{attribute addProperty BoxType "EK1100-0000-0018"}
{attribute addProperty Id "Beckhoff_EL72xxEK1122Beckhoff_EL72xxEK1122_DA7F4B70162A_0001_EL7201_0000_0017EL7201_83D4128E25031.25A_0002_EL7201_0000_0018EL7201_83D4128E25031.25A_0003_EL7201_0000_0019EL7201_83D4128E25031.25A_0004_EL7201_0000_0020EL7201_83D4128E25031.25A_0005_EL7201_0000_0021EL7201_83D4128E25031.25A_0006_EL7201_0001_0017EL7201_789C0F5925031.25A_0007_EL7201_0001_0018EL7201_789C0F5925031.25A_0008_EL7201_0001_0019EL7201_789C0F5925031.25A_0009_EL7201_0001_0020EL7201_789C0F5925031.25A_0010_EL7201_0001_0021EL7201_789C0F5925031.25A_0011_EL7201_0010_0019EL7201_83D4128E25031.25A_0012_EL7201_0010_0020EL7201_83D4128E25031.25A_0013_EL7201_0010_0021EL7201_83D4128E25031.25A_0014_EL7201_0010_0022EL7201_83D4128E25031.25A_0015_EL7201_0010_0023EL7201_83D4128E25031.25A_0016_EL7201_0010_0024EL7201_83D4128E25031.25A_0017_EL7201_0010_0025EL7201_83D4128E25031.25A_0018_EL7201_0010_0026EL7201_83D4128E25031.25A_0019_EL7201_0010_0027EL7201_83D4128E25031.25A_0020_EL7201_0010_0028EL7201_83D4128E25031.25A_0021_EL7201_0010_0029EL7201_83D4128E25031.25A_0022_EL7201_0010_0030EL7201_2D7B43DC25832.25A_0023_EL7201_0010_0031EL7201_2D7B43DC25832.25A_0024_EL7201_0010_0032EL7201_2D7B43DC25832.25A_0025_EL7201_0011_0019EL7201_789C0F5925031.25A_0026_EL7201_0011_0020EL7201_789C0F5925031.25A_0027_EL7201_0011_0021EL7201_789C0F5925031.25A_0028_EL7201_0011_0022EL7201_789C0F5925031.25A_0029_EL7201_0011_0023EL7201_789C0F5925031.25A_0030_EL7201_0011_0024EL7201_789C0F5925031.25A_0031_EL7201_0011_0025EL7201_789C0F5925031.25A_0032_EL7201_0011_0026EL7201_789C0F5925031.25A_0033_EL7201_0011_0027EL7201_789C0F5925031.25A_0034_EL7201_0011_0028EL7201_789C0F5925031.25A_0035_EL7201_0011_0029EL7201_789C0F5925031.25A_0036_EL7201_0011_0030EL7201_789C0F5925031.25A_0037_EL7201_0011_0031EL7201_789C0F5925031.25A_0038_EL7201_0011_0032EL7201_789C0F5925031.25A_0039_EL7211_0000_0020EL7211_83D4128E25031.25A_0040_EL7211_0000_0021EL7211_83D4128E25031.25A_0041_EL7211_0001_0020EL7211_789C0F5925031.25A_0042_EL7211_0001_0021EL7211_789C0F5925031.25A_0043_EL7211_0010_0023EL7211_83D4128E25031.25A_0044_EL7211_0010_0024EL7211_83D4128E25031.25A_0045_EL7211_0010_0025EL7211_83D4128E25031.25A_0046_EL7211_0010_0026EL7211_83D4128E25031.25A_0047_EL7211_0010_0027EL7211_83D4128E25031.25A_0048_EL7211_0010_0028EL7211_83D4128E25031.25A_0049_EL7211_0010_0029EL7211_83D4128E25031.25A_0050_EL7211_0010_0030EL7211_2D7B43DC25832.25A_0051_EL7211_0010_0031EL7211_2D7B43DC25832.25A_0052_EL7211_0010_0032EL7211_2D7B43DC25832.25A_0053_EL7211_0011_0023EL7211_789C0F5925031.25A_0054_EL7211_0011_0024EL7211_789C0F5925031.25A_0055_EL7211_0011_0025EL7211_789C0F5925031.25A_0056_EL7211_0011_0026EL7211_789C0F5925031.25A_0057_EL7211_0011_0027EL7211_789C0F5925031.25A_0058_EL7211_0011_0028EL7211_789C0F5925031.25A_0059_EL7211_0011_0029EL7211_789C0F5925031.25A_0060_EL7211_0011_0030EL7211_789C0F5925031.25A_0061_EL7211_0011_0031EL7211_789C0F5925031.25A_0062_EL7211_0011_0032EL7211_789C0F5925031.25A_0063_EL7201_9014_0026EL7201_83D4128E25031.25A_0064_EL7201_9014_0027EL7201_83D4128E25031.25A_0065_EL7201_9014_0028EL7201_83D4128E25031.25A_0066_EL7201_9014_0029EL7201_83D4128E25031.25A_0067_EL7201_9014_0030EL7201_2D7B43DC25832.25A_0068_EL7201_9014_0031EL7201_2D7B43DC25832.25A_0069_EL7201_9014_0032EL7201_2D7B43DC25832.25A_0070_EL7201_9015_0026EL7201_789C0F5925031.25A_0071_EL7201_9015_0027EL7201_789C0F5925031.25A_0072_EL7201_9015_0028EL7201_789C0F5925031.25A_0073_EL7201_9015_0029EL7201_789C0F5925031.25A_0074_EL7201_9015_0030EL7201_789C0F5925031.25A_0075_EL7201_9015_0031EL7201_789C0F5925031.25A_0076_EL7201_9015_0032EL7201_789C0F5925031.25A_0077_EL7211_9014_0026EL7211_83D4128E25031.25A_0078_EL7211_9014_0027EL7211_83D4128E25031.25A_0079_EL7211_9014_0028EL7211_83D4128E25031.25A_0080_EL7211_9014_0029EL7211_83D4128E25031.25A_0081_EL7211_9014_0030EL7211_2D7B43DC25832.25A_0082_EL7211_9014_0031EL7211_2D7B43DC25832.25A_0083_EL7211_9014_0032EL7211_2D7B43DC25832.25A_0084_EL7211_9015_0026EL7211_789C0F5925031.25A_0085_EL7211_9015_0027EL7211_789C0F5925031.25A_0086_EL7211_9015_0028EL7211_789C0F5925031.25A_0087_EL7211_9015_0029EL7211_789C0F5925031.25A_0088_EL7211_9015_0030EL7211_789C0F5925031.25A_0089_EL7211_9015_0031EL7211_789C0F5925031.25A_0090_EL7211_9015_0032EL7211_789C0F5925031.25A_0091_EL7221_0000_0021EL7221_83D4128E25031.25A_0092_EL7221_0001_0021EL7221_789C0F5925031.25A_0093_EL7221_9014_0028EL7221_83D4128E25031.25A_0094_EL7221_9014_0029EL7221_83D4128E25031.25A_0095_EL7221_9014_0030EL7221_2D7B43DC25832.25A_0096_EL7221_9014_0031EL7221_2D7B43DC25832.25A_0097_EL7221_9014_0032EL7221_2D7B43DC25832.25A_0098_EL7221_9015_0028EL7221_789C0F5925031.25A_0099_EL7221_9015_0029EL7221_789C0F5925031.25A_0100_EL7221_9015_0030EL7221_789C0F5925031.25A_0101_EL7221_9015_0031EL7221_789C0F5925031.25A_0102_EL7221_9015_0032EL7221_789C0F5925031.25"}
{attribute addProperty CRC "2978563334"}
{attribute addProperty SizeInBites "25636"}
{attribute addProperty SizeInBytes "3204.5"}
TYPE Beckhoff_EL72xx_B1894506 EXTENDS EK1100_179A0949 :
STRUCT
	{attribute addProperty Name "Beckhoff_EL72xxEK1122"}
	Beckhoff_EL72xxEK1122 : Beckhoff_EL72xxEK1122_DA7F4B70;
	{attribute addProperty Name "A_0001_EL7201_0000_0017"}
	A_0001_EL7201_0000_0017 : EL7201_83D4128E;
	{attribute addProperty Name "A_0002_EL7201_0000_0018"}
	A_0002_EL7201_0000_0018 : EL7201_83D4128E;
	{attribute addProperty Name "A_0003_EL7201_0000_0019"}
	A_0003_EL7201_0000_0019 : EL7201_83D4128E;
	{attribute addProperty Name "A_0004_EL7201_0000_0020"}
	A_0004_EL7201_0000_0020 : EL7201_83D4128E;
	{attribute addProperty Name "A_0005_EL7201_0000_0021"}
	A_0005_EL7201_0000_0021 : EL7201_83D4128E;
	{attribute addProperty Name "A_0006_EL7201_0001_0017"}
	A_0006_EL7201_0001_0017 : EL7201_789C0F59;
	{attribute addProperty Name "A_0007_EL7201_0001_0018"}
	A_0007_EL7201_0001_0018 : EL7201_789C0F59;
	{attribute addProperty Name "A_0008_EL7201_0001_0019"}
	A_0008_EL7201_0001_0019 : EL7201_789C0F59;
	{attribute addProperty Name "A_0009_EL7201_0001_0020"}
	A_0009_EL7201_0001_0020 : EL7201_789C0F59;
	{attribute addProperty Name "A_0010_EL7201_0001_0021"}
	A_0010_EL7201_0001_0021 : EL7201_789C0F59;
	{attribute addProperty Name "A_0011_EL7201_0010_0019"}
	A_0011_EL7201_0010_0019 : EL7201_83D4128E;
	{attribute addProperty Name "A_0012_EL7201_0010_0020"}
	A_0012_EL7201_0010_0020 : EL7201_83D4128E;
	{attribute addProperty Name "A_0013_EL7201_0010_0021"}
	A_0013_EL7201_0010_0021 : EL7201_83D4128E;
	{attribute addProperty Name "A_0014_EL7201_0010_0022"}
	A_0014_EL7201_0010_0022 : EL7201_83D4128E;
	{attribute addProperty Name "A_0015_EL7201_0010_0023"}
	A_0015_EL7201_0010_0023 : EL7201_83D4128E;
	{attribute addProperty Name "A_0016_EL7201_0010_0024"}
	A_0016_EL7201_0010_0024 : EL7201_83D4128E;
	{attribute addProperty Name "A_0017_EL7201_0010_0025"}
	A_0017_EL7201_0010_0025 : EL7201_83D4128E;
	{attribute addProperty Name "A_0018_EL7201_0010_0026"}
	A_0018_EL7201_0010_0026 : EL7201_83D4128E;
	{attribute addProperty Name "A_0019_EL7201_0010_0027"}
	A_0019_EL7201_0010_0027 : EL7201_83D4128E;
	{attribute addProperty Name "A_0020_EL7201_0010_0028"}
	A_0020_EL7201_0010_0028 : EL7201_83D4128E;
	{attribute addProperty Name "A_0021_EL7201_0010_0029"}
	A_0021_EL7201_0010_0029 : EL7201_83D4128E;
	{attribute addProperty Name "A_0022_EL7201_0010_0030"}
	A_0022_EL7201_0010_0030 : EL7201_2D7B43DC;
	{attribute addProperty Name "A_0023_EL7201_0010_0031"}
	A_0023_EL7201_0010_0031 : EL7201_2D7B43DC;
	{attribute addProperty Name "A_0024_EL7201_0010_0032"}
	A_0024_EL7201_0010_0032 : EL7201_2D7B43DC;
	{attribute addProperty Name "A_0025_EL7201_0011_0019"}
	A_0025_EL7201_0011_0019 : EL7201_789C0F59;
	{attribute addProperty Name "A_0026_EL7201_0011_0020"}
	A_0026_EL7201_0011_0020 : EL7201_789C0F59;
	{attribute addProperty Name "A_0027_EL7201_0011_0021"}
	A_0027_EL7201_0011_0021 : EL7201_789C0F59;
	{attribute addProperty Name "A_0028_EL7201_0011_0022"}
	A_0028_EL7201_0011_0022 : EL7201_789C0F59;
	{attribute addProperty Name "A_0029_EL7201_0011_0023"}
	A_0029_EL7201_0011_0023 : EL7201_789C0F59;
	{attribute addProperty Name "A_0030_EL7201_0011_0024"}
	A_0030_EL7201_0011_0024 : EL7201_789C0F59;
	{attribute addProperty Name "A_0031_EL7201_0011_0025"}
	A_0031_EL7201_0011_0025 : EL7201_789C0F59;
	{attribute addProperty Name "A_0032_EL7201_0011_0026"}
	A_0032_EL7201_0011_0026 : EL7201_789C0F59;
	{attribute addProperty Name "A_0033_EL7201_0011_0027"}
	A_0033_EL7201_0011_0027 : EL7201_789C0F59;
	{attribute addProperty Name "A_0034_EL7201_0011_0028"}
	A_0034_EL7201_0011_0028 : EL7201_789C0F59;
	{attribute addProperty Name "A_0035_EL7201_0011_0029"}
	A_0035_EL7201_0011_0029 : EL7201_789C0F59;
	{attribute addProperty Name "A_0036_EL7201_0011_0030"}
	A_0036_EL7201_0011_0030 : EL7201_789C0F59;
	{attribute addProperty Name "A_0037_EL7201_0011_0031"}
	A_0037_EL7201_0011_0031 : EL7201_789C0F59;
	{attribute addProperty Name "A_0038_EL7201_0011_0032"}
	A_0038_EL7201_0011_0032 : EL7201_789C0F59;
	{attribute addProperty Name "A_0039_EL7211_0000_0020"}
	A_0039_EL7211_0000_0020 : EL7211_83D4128E;
	{attribute addProperty Name "A_0040_EL7211_0000_0021"}
	A_0040_EL7211_0000_0021 : EL7211_83D4128E;
	{attribute addProperty Name "A_0041_EL7211_0001_0020"}
	A_0041_EL7211_0001_0020 : EL7211_789C0F59;
	{attribute addProperty Name "A_0042_EL7211_0001_0021"}
	A_0042_EL7211_0001_0021 : EL7211_789C0F59;
	{attribute addProperty Name "A_0043_EL7211_0010_0023"}
	A_0043_EL7211_0010_0023 : EL7211_83D4128E;
	{attribute addProperty Name "A_0044_EL7211_0010_0024"}
	A_0044_EL7211_0010_0024 : EL7211_83D4128E;
	{attribute addProperty Name "A_0045_EL7211_0010_0025"}
	A_0045_EL7211_0010_0025 : EL7211_83D4128E;
	{attribute addProperty Name "A_0046_EL7211_0010_0026"}
	A_0046_EL7211_0010_0026 : EL7211_83D4128E;
	{attribute addProperty Name "A_0047_EL7211_0010_0027"}
	A_0047_EL7211_0010_0027 : EL7211_83D4128E;
	{attribute addProperty Name "A_0048_EL7211_0010_0028"}
	A_0048_EL7211_0010_0028 : EL7211_83D4128E;
	{attribute addProperty Name "A_0049_EL7211_0010_0029"}
	A_0049_EL7211_0010_0029 : EL7211_83D4128E;
	{attribute addProperty Name "A_0050_EL7211_0010_0030"}
	A_0050_EL7211_0010_0030 : EL7211_2D7B43DC;
	{attribute addProperty Name "A_0051_EL7211_0010_0031"}
	A_0051_EL7211_0010_0031 : EL7211_2D7B43DC;
	{attribute addProperty Name "A_0052_EL7211_0010_0032"}
	A_0052_EL7211_0010_0032 : EL7211_2D7B43DC;
	{attribute addProperty Name "A_0053_EL7211_0011_0023"}
	A_0053_EL7211_0011_0023 : EL7211_789C0F59;
	{attribute addProperty Name "A_0054_EL7211_0011_0024"}
	A_0054_EL7211_0011_0024 : EL7211_789C0F59;
	{attribute addProperty Name "A_0055_EL7211_0011_0025"}
	A_0055_EL7211_0011_0025 : EL7211_789C0F59;
	{attribute addProperty Name "A_0056_EL7211_0011_0026"}
	A_0056_EL7211_0011_0026 : EL7211_789C0F59;
	{attribute addProperty Name "A_0057_EL7211_0011_0027"}
	A_0057_EL7211_0011_0027 : EL7211_789C0F59;
	{attribute addProperty Name "A_0058_EL7211_0011_0028"}
	A_0058_EL7211_0011_0028 : EL7211_789C0F59;
	{attribute addProperty Name "A_0059_EL7211_0011_0029"}
	A_0059_EL7211_0011_0029 : EL7211_789C0F59;
	{attribute addProperty Name "A_0060_EL7211_0011_0030"}
	A_0060_EL7211_0011_0030 : EL7211_789C0F59;
	{attribute addProperty Name "A_0061_EL7211_0011_0031"}
	A_0061_EL7211_0011_0031 : EL7211_789C0F59;
	{attribute addProperty Name "A_0062_EL7211_0011_0032"}
	A_0062_EL7211_0011_0032 : EL7211_789C0F59;
	{attribute addProperty Name "A_0063_EL7201_9014_0026"}
	A_0063_EL7201_9014_0026 : EL7201_83D4128E;
	{attribute addProperty Name "A_0064_EL7201_9014_0027"}
	A_0064_EL7201_9014_0027 : EL7201_83D4128E;
	{attribute addProperty Name "A_0065_EL7201_9014_0028"}
	A_0065_EL7201_9014_0028 : EL7201_83D4128E;
	{attribute addProperty Name "A_0066_EL7201_9014_0029"}
	A_0066_EL7201_9014_0029 : EL7201_83D4128E;
	{attribute addProperty Name "A_0067_EL7201_9014_0030"}
	A_0067_EL7201_9014_0030 : EL7201_2D7B43DC;
	{attribute addProperty Name "A_0068_EL7201_9014_0031"}
	A_0068_EL7201_9014_0031 : EL7201_2D7B43DC;
	{attribute addProperty Name "A_0069_EL7201_9014_0032"}
	A_0069_EL7201_9014_0032 : EL7201_2D7B43DC;
	{attribute addProperty Name "A_0070_EL7201_9015_0026"}
	A_0070_EL7201_9015_0026 : EL7201_789C0F59;
	{attribute addProperty Name "A_0071_EL7201_9015_0027"}
	A_0071_EL7201_9015_0027 : EL7201_789C0F59;
	{attribute addProperty Name "A_0072_EL7201_9015_0028"}
	A_0072_EL7201_9015_0028 : EL7201_789C0F59;
	{attribute addProperty Name "A_0073_EL7201_9015_0029"}
	A_0073_EL7201_9015_0029 : EL7201_789C0F59;
	{attribute addProperty Name "A_0074_EL7201_9015_0030"}
	A_0074_EL7201_9015_0030 : EL7201_789C0F59;
	{attribute addProperty Name "A_0075_EL7201_9015_0031"}
	A_0075_EL7201_9015_0031 : EL7201_789C0F59;
	{attribute addProperty Name "A_0076_EL7201_9015_0032"}
	A_0076_EL7201_9015_0032 : EL7201_789C0F59;
	{attribute addProperty Name "A_0077_EL7211_9014_0026"}
	A_0077_EL7211_9014_0026 : EL7211_83D4128E;
	{attribute addProperty Name "A_0078_EL7211_9014_0027"}
	A_0078_EL7211_9014_0027 : EL7211_83D4128E;
	{attribute addProperty Name "A_0079_EL7211_9014_0028"}
	A_0079_EL7211_9014_0028 : EL7211_83D4128E;
	{attribute addProperty Name "A_0080_EL7211_9014_0029"}
	A_0080_EL7211_9014_0029 : EL7211_83D4128E;
	{attribute addProperty Name "A_0081_EL7211_9014_0030"}
	A_0081_EL7211_9014_0030 : EL7211_2D7B43DC;
	{attribute addProperty Name "A_0082_EL7211_9014_0031"}
	A_0082_EL7211_9014_0031 : EL7211_2D7B43DC;
	{attribute addProperty Name "A_0083_EL7211_9014_0032"}
	A_0083_EL7211_9014_0032 : EL7211_2D7B43DC;
	{attribute addProperty Name "A_0084_EL7211_9015_0026"}
	A_0084_EL7211_9015_0026 : EL7211_789C0F59;
	{attribute addProperty Name "A_0085_EL7211_9015_0027"}
	A_0085_EL7211_9015_0027 : EL7211_789C0F59;
	{attribute addProperty Name "A_0086_EL7211_9015_0028"}
	A_0086_EL7211_9015_0028 : EL7211_789C0F59;
	{attribute addProperty Name "A_0087_EL7211_9015_0029"}
	A_0087_EL7211_9015_0029 : EL7211_789C0F59;
	{attribute addProperty Name "A_0088_EL7211_9015_0030"}
	A_0088_EL7211_9015_0030 : EL7211_789C0F59;
	{attribute addProperty Name "A_0089_EL7211_9015_0031"}
	A_0089_EL7211_9015_0031 : EL7211_789C0F59;
	{attribute addProperty Name "A_0090_EL7211_9015_0032"}
	A_0090_EL7211_9015_0032 : EL7211_789C0F59;
	{attribute addProperty Name "A_0091_EL7221_0000_0021"}
	A_0091_EL7221_0000_0021 : EL7221_83D4128E;
	{attribute addProperty Name "A_0092_EL7221_0001_0021"}
	A_0092_EL7221_0001_0021 : EL7221_789C0F59;
	{attribute addProperty Name "A_0093_EL7221_9014_0028"}
	A_0093_EL7221_9014_0028 : EL7221_83D4128E;
	{attribute addProperty Name "A_0094_EL7221_9014_0029"}
	A_0094_EL7221_9014_0029 : EL7221_83D4128E;
	{attribute addProperty Name "A_0095_EL7221_9014_0030"}
	A_0095_EL7221_9014_0030 : EL7221_2D7B43DC;
	{attribute addProperty Name "A_0096_EL7221_9014_0031"}
	A_0096_EL7221_9014_0031 : EL7221_2D7B43DC;
	{attribute addProperty Name "A_0097_EL7221_9014_0032"}
	A_0097_EL7221_9014_0032 : EL7221_2D7B43DC;
	{attribute addProperty Name "A_0098_EL7221_9015_0028"}
	A_0098_EL7221_9015_0028 : EL7221_789C0F59;
	{attribute addProperty Name "A_0099_EL7221_9015_0029"}
	A_0099_EL7221_9015_0029 : EL7221_789C0F59;
	{attribute addProperty Name "A_0100_EL7221_9015_0030"}
	A_0100_EL7221_9015_0030 : EL7221_789C0F59;
	{attribute addProperty Name "A_0101_EL7221_9015_0031"}
	A_0101_EL7221_9015_0031 : EL7221_789C0F59;
	{attribute addProperty Name "A_0102_EL7221_9015_0032"}
	A_0102_EL7221_9015_0032 : EL7221_789C0F59;
END_STRUCT
END_TYPE

(* stored: Version 1.2.0.0, ProductVersion 3.1.4024.9
   DUT Beckhoff_EL72xx_B1894506: Id {5f2a7588-87b9-43a8-91c8-1ab2dc57ed92} *)
